FUNCTION_BLOCK FB_Tail
VAR_INPUT
	sMessage1 :T_MaxString;
	sMessage2 :T_MaxString;
	sMessage3 :T_MaxString;
	sMessage4 :T_MaxString;
    bReset:BOOL;
END_VAR
VAR_OUTPUT
	
	
END_VAR
VAR
	fbBuffer:FB_TransBuffer;
	aTransBuff : ARRAY[1..10] OF T_MaxString;
	
	bReady:BOOL;
	bEmpty:BOOL;
END_VAR
VAR_IN_OUT
	bMessageReady1:BOOL;
	bMessageReady2:BOOL;
	bMessageReady3:BOOL;
	bMessageReady4:BOOL;
	bShiftBuff:BOOL;
	sMessageOut:T_MaxString;
	bNew:BOOL;
END_VAR


IF bMessageReady1 AND NOT fbBuffer.bBusy  THEN
	fbBuffer(sTrans:=sMessage1,bWriteInBuff:=bMessageReady1,aTransBuff:=aTransBuff,bShiftBuff:=bShiftBuff,bNew:=bNew);
END_IF
IF bMessageReady2 AND NOT fbBuffer.bBusy  THEN
	fbBuffer(sTrans:=sMessage2,bWriteInBuff:=bMessageReady2,aTransBuff:=aTransBuff,bShiftBuff:=bShiftBuff,bNew:=bNew);
END_IF
IF bMessageReady3 AND NOT fbBuffer.bBusy  THEN
	fbBuffer(sTrans:=sMessage3,bWriteInBuff:=bMessageReady3,aTransBuff:=aTransBuff,bShiftBuff:=bShiftBuff,bNew:=bNew);
END_IF
IF bMessageReady4 AND NOT fbBuffer.bBusy  THEN
	fbBuffer(sTrans:=sMessage4,bWriteInBuff:=bMessageReady4,aTransBuff:=aTransBuff,bShiftBuff:=bShiftBuff,bNew:=bNew);
END_IF





(*
IF bMessageReady1 AND NOT fbBuffer.bBusy  THEN
	fbBuffer(sTrans:=sMessage1,bWriteInBuff:=bMessageReady1,aTransBuff:=aTransBuff,bShiftBuff:=bShiftBuff);
   IF	NOT fbBuffer.bBusy THEN
	   bReady:=TRUE;
   END_IF
   
   
   
ELSIF bMessageReady2 AND NOT fbBuffer.bBusy THEN
	fbBuffer(sTrans:=sMessage2,bWriteInBuff:=bMessageReady2,aTransBuff:=aTransBuff,bShiftBuff:=bShiftBuff);
	  IF	NOT fbBuffer.bBusy THEN
	   bReady:=TRUE;
   END_IF 
ELSIF bMessageReady3 THEN
	fbBuffer(sTrans:=sMessage3,bWriteInBuff:=bMessageReady3,aTransBuff:=aTransBuff,bShiftBuff:=bShiftBuff);	
ELSIF bMessageReady4 THEN
	fbBuffer(sTrans:=sMessage4,bWriteInBuff:=bMessageReady4,aTransBuff:=aTransBuff,bShiftBuff:=bShiftBuff);	
	*)
	
(*IF 	NOT fbBuffer.bBusy  THEN
	fbBuffer(sTrans:=sMessage1,bWriteInBuff:=bMessageReady1,aTransBuff:=aTransBuff,bShiftBuff:=bEmpty);
	fbBuffer(sTrans:=sMessage2,bWriteInBuff:=bMessageReady2,aTransBuff:=aTransBuff,bShiftBuff:=bEmpty);
    fbBuffer(sTrans:=sMessage3,bWriteInBuff:=bMessageReady3,aTransBuff:=aTransBuff,bShiftBuff:=bEmpty);	
    fbBuffer(sTrans:=sMessage4,bWriteInBuff:=bMessageReady4,aTransBuff:=aTransBuff,bShiftBuff:=bEmpty);	
    fbBuffer(bWriteInBuff:=bEmpty,aTransBuff:=aTransBuff,bShiftBuff:=bShiftBuff);
END_IF*)
	
   fbBuffer(bWriteInBuff:=bEmpty,aTransBuff:=aTransBuff,bShiftBuff:=bShiftBuff,bReset:=bReset,bNew:=bNew);
   
	sMessageOut:=fbBuffer.sTransBuffOut;

END_FUNCTION_BLOCK

(* stored: Version 1.1.0.1, ProductVersion 3.1.4024.4
   POU FB_Tail: Id {4cea5162-f671-492a-a4d3-4e7dfbed35c7}, SpecialFunc None *)
